TYPE ST_DOX_Control :
STRUCT
	bBit0    :				BIT;	//71.0
	bBit1    :				BIT;
	bBit2    :				BIT;
	bPWM  :					BIT:=1;	//71.3
	bBit4  :				BIT;
	bBit5  :				BIT;
	bBit6  :				BIT;
	bReset  :				BIT;	//71.7
	BByte8   :				BYTE;
	
END_STRUCT
END_TYPE

(* stored: Version 1.1.0.1, ProductVersion 3.1.4019.2
   DUT ST_DOX_Control: Id {a08930eb-15b6-4eaa-b623-7c9c3b818f19} *)
